TYPE ST_HardSettings_DCcharger :
STRUCT
	r_PowerMax			: REAL;
END_STRUCT
END_TYPE

(* stored: Version 1.1.0.1, ProductVersion 3.1.4026.18
   DUT ST_HardSettings_DCcharger: Id {2f92fac2-7ed7-4d50-b4ab-7b9f6a582359} *)
